# EPICS autosave request: quadEMApp/Db/FX4_settings.req
$(P)$(R)CurrentUnits
